PROGRAM MainCtrl
VAR
	ForceFan1: aFb_Motor;
	ForceFan2: aFb_Motor;
	ForceFan3: aFb_Motor;
	CondensePump: aFb_Motor;
	SupplyPump: aFb_Motor;
	CircularPump: aFb_Motor;
	
	ForceFan1_PID: FB_BasicPID;
	ForceFan2_PID: FB_BasicPID;
	ForceFan3_PID: FB_BasicPID;
	CondensePump_PID: FB_BasicPID;
	SupplyPump_PID: FB_BasicPID;
	CircularPump_PID: FB_BasicPID;

	start: BOOL;
	stop: BOOL;
	setpoint: LREAL := 0.266;
	setpoint2: LREAL := 28;
	setpoint3: LREAL := 167;
	setpoint4: LREAL := 1350;
END_VAR

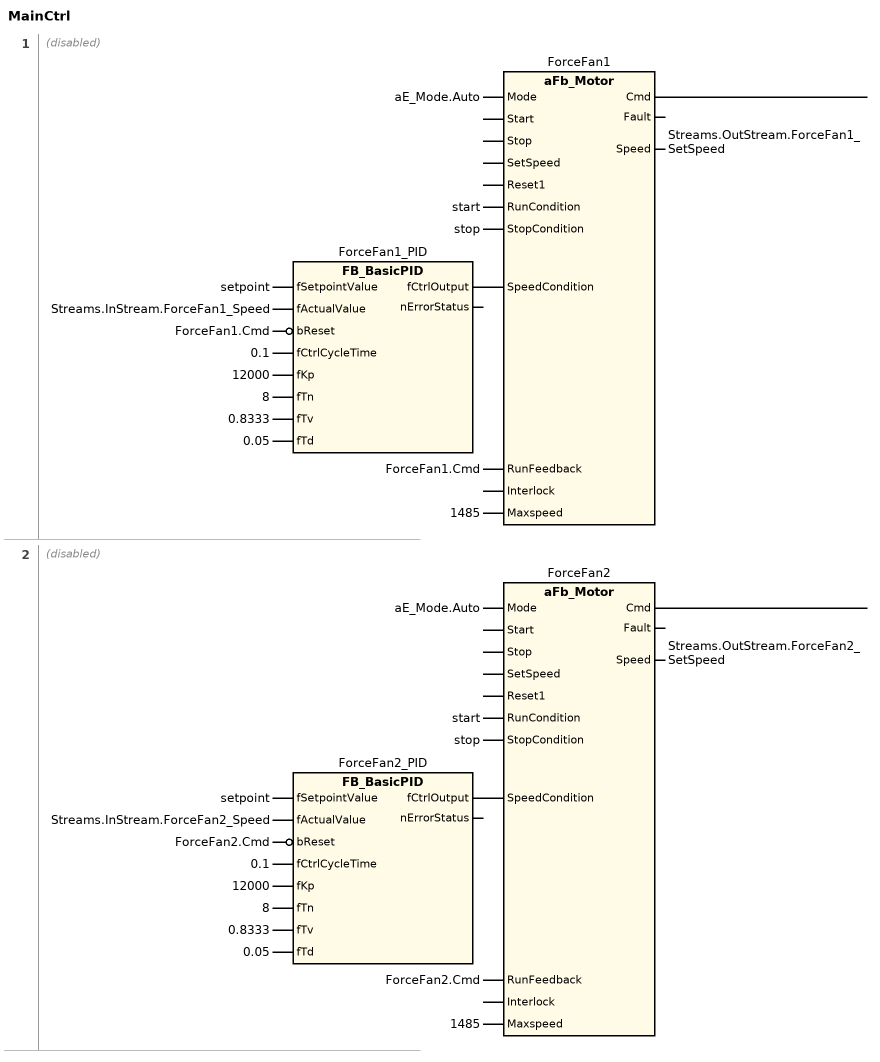
// NETWORK 1 (disabled)
// ForceFan1_PID(
//     fSetpointValue := setpoint,
//     fActualValue := Streams.InStream.ForceFan1_Speed,
//     bReset := NOT ForceFan1.Cmd,
//     fCtrlCycleTime := 0.1,
//     fKp := 12000,
//     fTn := 8,
//     fTv := 0.8333,
//     fTd := 0.05); // FB_BasicPID
// ForceFan1(
//     Mode := aE_Mode.Auto,
//     RunCondition := start,
//     StopCondition := stop,
//     SpeedCondition := ForceFan1_PID.fCtrlOutput,
//     RunFeedback := ForceFan1.Cmd,
//     Maxspeed := 1485,
//     Speed => Streams.OutStream.ForceFan1_SetSpeed); // aFb_Motor

// NETWORK 2 (disabled)
// ForceFan2_PID(
//     fSetpointValue := setpoint,
//     fActualValue := Streams.InStream.ForceFan2_Speed,
//     bReset := NOT ForceFan2.Cmd,
//     fCtrlCycleTime := 0.1,
//     fKp := 12000,
//     fTn := 8,
//     fTv := 0.8333,
//     fTd := 0.05); // FB_BasicPID
// ForceFan2(
//     Mode := aE_Mode.Auto,
//     RunCondition := start,
//     StopCondition := stop,
//     SpeedCondition := ForceFan2_PID.fCtrlOutput,
//     RunFeedback := ForceFan2.Cmd,
//     Maxspeed := 1485,
//     Speed => Streams.OutStream.ForceFan2_SetSpeed); // aFb_Motor

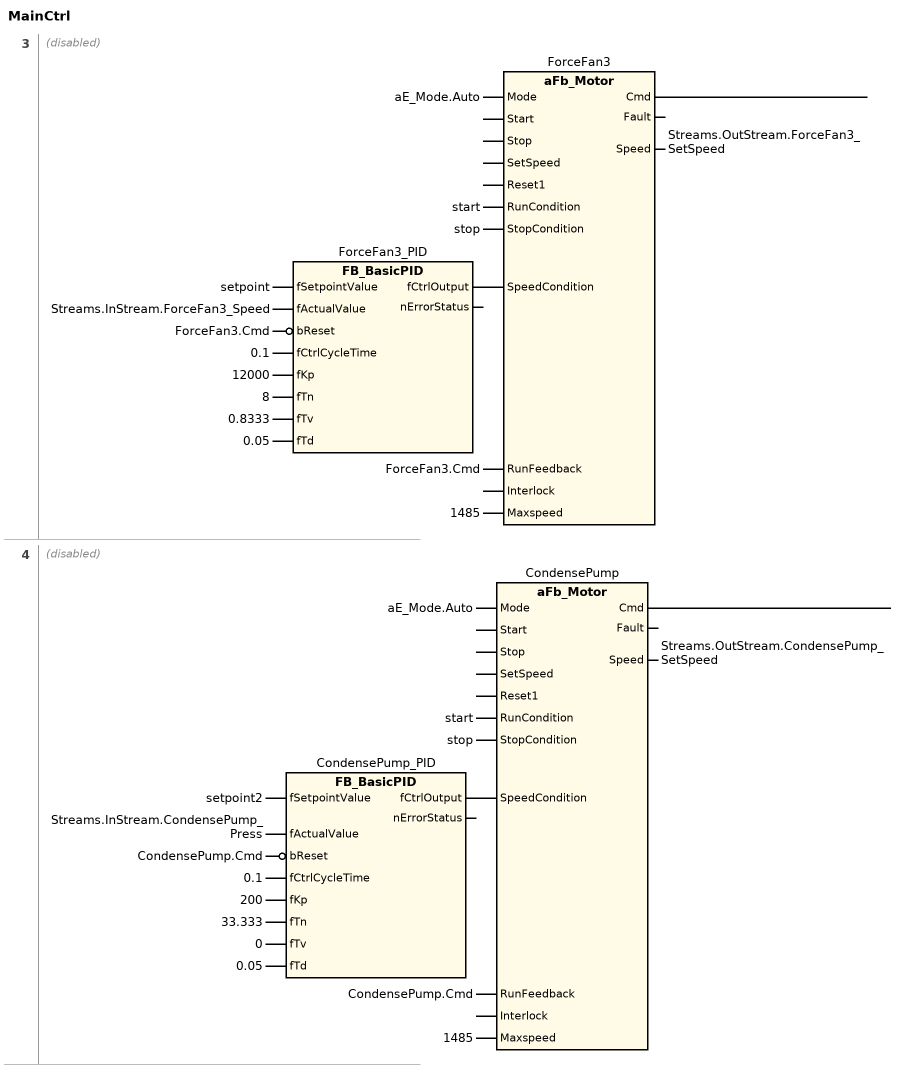
// NETWORK 3 (disabled)
// ForceFan3_PID(
//     fSetpointValue := setpoint,
//     fActualValue := Streams.InStream.ForceFan3_Speed,
//     bReset := NOT ForceFan3.Cmd,
//     fCtrlCycleTime := 0.1,
//     fKp := 12000,
//     fTn := 8,
//     fTv := 0.8333,
//     fTd := 0.05); // FB_BasicPID
// ForceFan3(
//     Mode := aE_Mode.Auto,
//     RunCondition := start,
//     StopCondition := stop,
//     SpeedCondition := ForceFan3_PID.fCtrlOutput,
//     RunFeedback := ForceFan3.Cmd,
//     Maxspeed := 1485,
//     Speed => Streams.OutStream.ForceFan3_SetSpeed); // aFb_Motor

// NETWORK 4 (disabled)
// CondensePump_PID(
//     fSetpointValue := setpoint2,
//     fActualValue := Streams.InStream.CondensePump_Press,
//     bReset := NOT CondensePump.Cmd,
//     fCtrlCycleTime := 0.1,
//     fKp := 200,
//     fTn := 33.333,
//     fTv := 0,
//     fTd := 0.05); // FB_BasicPID
// CondensePump(
//     Mode := aE_Mode.Auto,
//     RunCondition := start,
//     StopCondition := stop,
//     SpeedCondition := CondensePump_PID.fCtrlOutput,
//     RunFeedback := CondensePump.Cmd,
//     Maxspeed := 1485,
//     Speed => Streams.OutStream.CondensePump_SetSpeed); // aFb_Motor

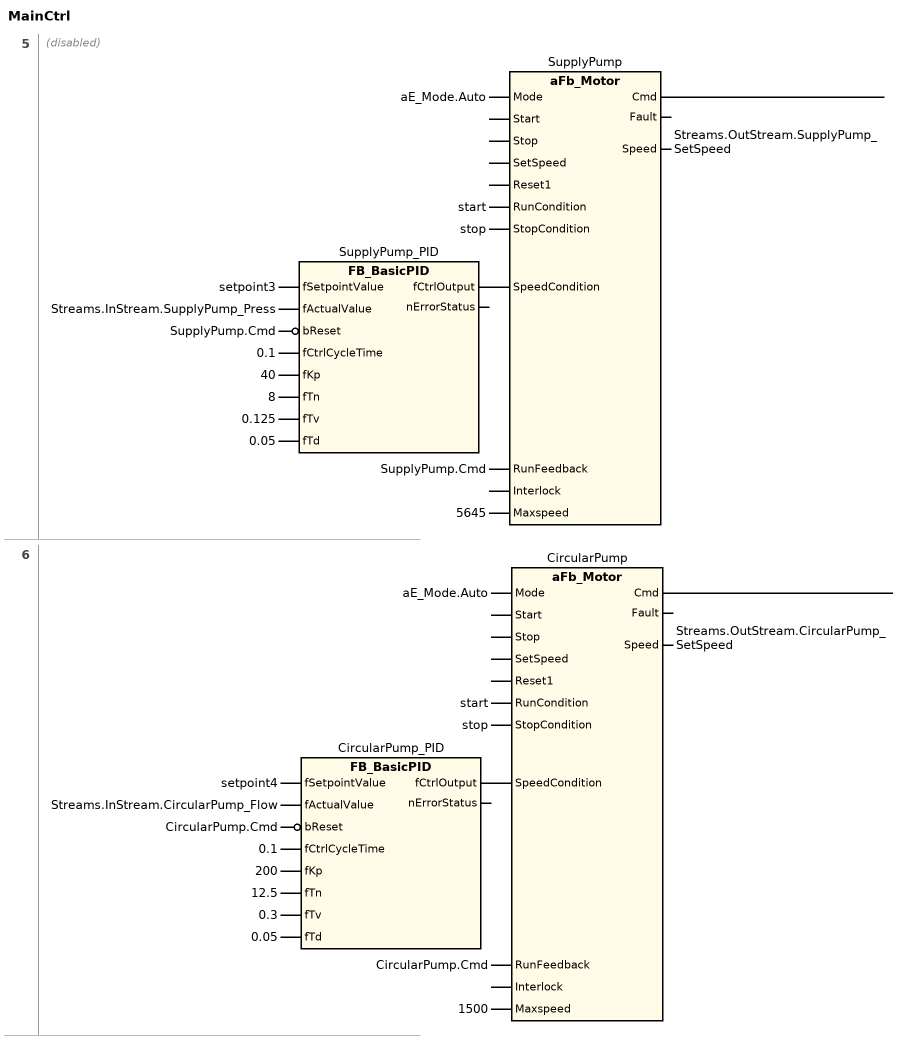
// NETWORK 5 (disabled)
// SupplyPump_PID(
//     fSetpointValue := setpoint3,
//     fActualValue := Streams.InStream.SupplyPump_Press,
//     bReset := NOT SupplyPump.Cmd,
//     fCtrlCycleTime := 0.1,
//     fKp := 40,
//     fTn := 8,
//     fTv := 0.125,
//     fTd := 0.05); // FB_BasicPID
// SupplyPump(
//     Mode := aE_Mode.Auto,
//     RunCondition := start,
//     StopCondition := stop,
//     SpeedCondition := SupplyPump_PID.fCtrlOutput,
//     RunFeedback := SupplyPump.Cmd,
//     Maxspeed := 5645,
//     Speed => Streams.OutStream.SupplyPump_SetSpeed); // aFb_Motor

// NETWORK 6
CircularPump_PID(
    fSetpointValue := setpoint4,
    fActualValue := Streams.InStream.CircularPump_Flow,
    bReset := NOT CircularPump.Cmd,
    fCtrlCycleTime := 0.1,
    fKp := 200,
    fTn := 12.5,
    fTv := 0.3,
    fTd := 0.05); // FB_BasicPID
CircularPump(
    Mode := aE_Mode.Auto,
    RunCondition := start,
    StopCondition := stop,
    SpeedCondition := CircularPump_PID.fCtrlOutput,
    RunFeedback := CircularPump.Cmd,
    Maxspeed := 1500,
    Speed => Streams.OutStream.CircularPump_SetSpeed); // aFb_Motor

END_PROGRAM

(* stored: Version 1.1.0.1, ProductVersion 3.1.4024.4
   POU MainCtrl: Id {686e13a1-eb41-45b3-a154-fe93b25c8d73}, SpecialFunc None *)
